// TIA Portal V20 export
TYPE "SEW_MOVIKIT_VelocityDrive_SETPOINTS_V2.1"
   STRUCT
      x_Bit_8_Fault_Reset : Bool;
      x_Bit_9_Reserved : Bool;
      x_Bit_10_Activate_DriveTrain2 : Bool;
      x_Bit_11_Reserved : Bool;
      x_Bit_12_Deactivate_SW_Limit_switches : Bool;
      x_Bit_13_Activate_Output_Stage_Inhibit : Bool;
      x_Bit_14_Activate_StandBy_Mode : Bool;
      x_Bit_15_Heartbeat_IN : Bool;
      x_Bit_0_Enable_Emergency_Stop : Bool;
      x_Bit_1_Enable_Application_Stop : Bool;
      x_Bit_2_Reserved : Bool;
      x_Bit_3_Release_Brake : Bool;
      x_Bit_4_Jog_positive : Bool;
      x_Bit_5_Jog_negative : Bool;
      x_Bit_6_Apply_relative_Position : Bool;
      x_Bit_7_Start_Stop : Bool;
      iSetpoint_Speed : Int;
      iSetpoint_Acceleration : Int;
      iSetpoint_Deceleration : Int;
      wDigital_Outputs : Word;
   END_STRUCT;
END_TYPE
